{attribute 'linkalways'} 
{attribute 'no_explicit_call' := 'This FB is a CLASS and must be accessed using methods or properties'}
{attribute 'enable_dynamic_creation'}
FUNCTION_BLOCK Node_F_VN_AppendToContainer_TcVnVector3_REAL EXTENDS VisionNode
VAR
    aElement : _TcVnVector3_REAL;
    ipContainer : _ITcVnContainer;
    hrPrev : _HRESULT(S_OK);
	hresult : _HRESULT(S_OK);
END_VAR

METHOD PUBLIC  Clone : I_Node
VAR
	pNode : POINTER TO Node_F_VN_AppendToContainer_TcVnVector3_REAL;
END_VAR
pNode := __NEW(Node_F_VN_AppendToContainer_TcVnVector3_REAL);
Clone := pNode^;
END_METHOD

METHOD FB_init : BOOL
VAR_INPUT
	bInitRetains : BOOL; // if TRUE, the retain variables are initialized (warm start / cold start)
	bInCopyCode : BOOL;  // if TRUE, the instance afterwards gets moved into the copy code (online change)
END_VAR
AddInput('aElement', aElement);
AddInput('ipContainer', ipContainer);
AddInput('hrPrev', hrPrev);
AddOutput('ipContainer', ipContainer);
AddOutput('hresult',hresult);
END_METHOD

METHOD PROTECTED OnExecute : HRESULT
hresult.Value := F_VN_AppendToContainer_TcVnVector3_REAL(
    aElement := aElement.Value,
	ipContainer := ipContainer.Value,
	hrPrev:= hrPrev.Value);
END_METHOD

METHOD PUBLIC PreExecutionCheck
VAR_INPUT
	Check : I_PreExecutionChecks;
END_VAR
Check.IsTrue(ipContainer.IsValid, 'ipContainer must be a valid container');
END_METHOD

END_FUNCTION_BLOCK

(* stored: Version 1.1.0.1, ProductVersion 3.1.4024.13
   POU Node_F_VN_AppendToContainer_TcVnVector3_REAL: Id {a19cf258-64e5-4da0-9fe1-d4fdcfd44012}, SpecialFunc None
   Folder Constructor: Id {7b63501e-531f-4afe-b39a-d13f3e795c76}
   Method Clone: Id {f500f0f6-9bb3-4964-bad2-515d8e06b882}
   Method FB_init: Id {89e45bab-1472-498e-9c89-b617780d7027}
   Method OnExecute: Id {3f289863-9009-4acc-92fd-80c84259768b}
   Method PreExecutionCheck: Id {2d98a7b9-e98e-41ee-a9dc-9da8747c1499} *)
